PROGRAM PRG_SFLX_03_AddtitionalConvCtrl
VAR
	fbAddtitionalConvDelay	 : FB_TOFR;
END_VAR

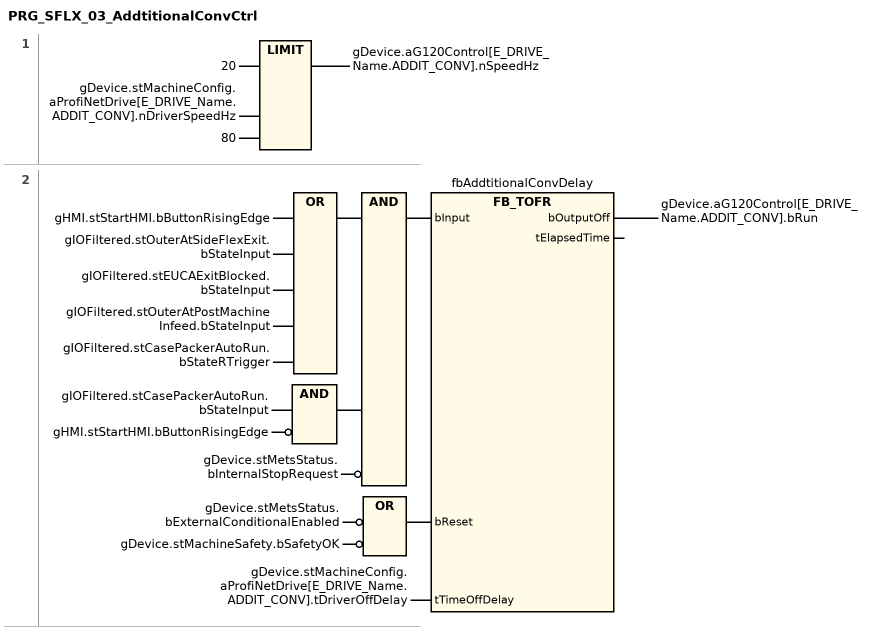
// NETWORK 1
gDevice.aG120Control[E_DRIVE_Name.ADDIT_CONV].nSpeedHz := LIMIT(20, gDevice.stMachineConfig.aProfiNetDrive[E_DRIVE_Name.ADDIT_CONV].nDriverSpeedHz, 80);

// NETWORK 2
fbAddtitionalConvDelay(
    bInput := (gHMI.stStartHMI.bButtonRisingEdge OR gIOFiltered.stOuterAtSideFlexExit.bStateInput OR gIOFiltered.stEUCAExitBlocked.bStateInput OR gIOFiltered.stOuterAtPostMachineInfeed.bStateInput OR gIOFiltered.stCasePackerAutoRun.bStateRTrigger) AND (gIOFiltered.stCasePackerAutoRun.bStateInput AND NOT gHMI.stStartHMI.bButtonRisingEdge) AND NOT gDevice.stMetsStatus.bInternalStopRequest,
    bReset := NOT gDevice.stMetsStatus.bExternalConditionalEnabled OR NOT gDevice.stMachineSafety.bSafetyOK,
    tTimeOffDelay := gDevice.stMachineConfig.aProfiNetDrive[E_DRIVE_Name.ADDIT_CONV].tDriverOffDelay); // FB_TOFR
gDevice.aG120Control[E_DRIVE_Name.ADDIT_CONV].bRun := fbAddtitionalConvDelay.bOutputOff;

END_PROGRAM

(* stored: Version 1.1.0.1
   POU PRG_SFLX_03_AddtitionalConvCtrl: Id {892ddcf1-3b83-4a22-8a65-a2864c2f037a}, SpecialFunc None *)
